TYPE TcaSafetyGateStatus :
STRUCT
    ActionDescription : STRING(100);	         
	Safe : BOOL;
	Open : BOOL;
	ComponentsAreService : BOOL;
	
END_STRUCT
END_TYPE

(* stored: Version 1.1.0.1
   DUT TcaSafetyGateStatus: Id {b3c2906d-08a9-45c4-88dc-9922739a3d6a} *)
